// TIA Portal V20 export
DATA_BLOCK "InstTorqueCal_TopTapeAxisX"   // DB338
// stored: AssignedProDiagFB ProDiag, InstanceOfName LER_ServoTorqueCal, InstanceOfType FB
"LER_ServoTorqueCal"
   // VAR_INPUT
   //    enable : Bool;
   //    enableManualCmds : Bool;
   //    storageCount : UInt;
   //    storageCycle : Bool;
   //    RatedTorque : LReal;
   //    axis : DB_ANY;
   // END_VAR
   // VAR_OUTPUT
   //    actualTorque : LReal;
   //    averageTorque : LReal;
   //    peakTorque : LReal;
   //    currentload : LReal;
   //    averageload : LReal;
   //    peakload : LReal;
   // END_VAR
   // VAR_IN_OUT
   //    configuration : "LER_typeServoTorqueCalConfigruation";
   //    moduleInterface : "LER_typeServoTorqueCalInterface";
   // END_VAR
   // VAR
   //    statTonTimer : Array[0..9] of TON_TIME;
   //    statCurrentTorqueDataBuf : Array[0..99] of LReal;
   //    statPulse : Array[0..9] of Bool;
   //    statActualTorque : LReal;
   //    statAverageTorque : LReal;
   //    statPeakTorque : LReal;
   //    statActualLoad : LReal;
   //    statAverageLoad : LReal;
   //    statPeakLoad : LReal;
   //    statMoveCount : UInt;
   //    statResetCmd : Bool;
   //    statOverloadWarning : Bool;
   //    statOverloadAlarm : Bool;
   // END_VAR
BEGIN
END_DATA_BLOCK
